{attribute 'reflection'} 
FUNCTION_BLOCK FB_IPCDiagnostics IMPLEMENTS I_SysModules
VAR
	nCpuTemperature	: INT := 75;	// CPU temperature [°F]
	nCpuUsage       : INT := 5;    // CPU usage [%]
	
	
	{attribute 'instance-path'} 
    {attribute 'noinit'} 
    sPath : STRING; 
END_VAR

METHOD accept
VAR_INPUT
	iVisitor : I_Visitor;
END_VAR
iVisitor.visitIPC(THIS^);
END_METHOD

PROPERTY pCPU_Temp : INT
GET
pCPU_Temp := THIS^.nCpuTemperature;
END_GET
END_PROPERTY

PROPERTY pCPU_Usage : INT
GET
pCPU_Usage := THIS^.nCpuUsage;
END_GET
END_PROPERTY

PROPERTY pPath : STRING
GET
pPath := THIS^.sPath;
END_GET
END_PROPERTY

END_FUNCTION_BLOCK

(* stored: Version 1.1.0.1, ProductVersion 3.1.4024.12
   POU FB_IPCDiagnostics: Id {03aa6bb3-78ca-4569-b572-44f1a01ac209}, SpecialFunc None
   Method accept: Id {dea57fa9-4cb0-49ab-b208-c1b1b2cddc11}
   Property pCPU_Temp: Id {472bdcca-bfb7-47fc-a956-db1deb7ad691}
   Get Get: Id {d9b06717-4643-4732-974c-328779b5900a}
   Property pCPU_Usage: Id {2a4155f8-1d71-414c-bdd2-b4128803e0a8}
   Get Get: Id {ff853849-7244-4797-a537-981cf8960313}
   Property pPath: Id {a7b72c3a-26f7-4006-8cf0-41ee057228c4}
   Get Get: Id {aa052426-48ed-4e7a-b213-8a3e9a5f0b93} *)
